FUNCTION_BLOCK Stage13 (* Template for a Basic Function Block Type *)
  (* Standard: 61499-2 *)
  (* Version 1.0, 2021-06-20, HP *)
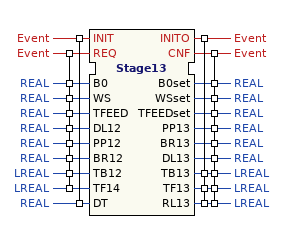
  EVENT_INPUT
    INIT WITH DT; (* Initialization Request *)
    REQ WITH B0, WS, TFEED, DL12, PP12, BR12, TB12, TF14; (* Normal Execution Request *)
  END_EVENT
  EVENT_OUTPUT
    INITO WITH TB13, TF13, RL13; (* Initialization Confirm *)
    CNF WITH TB13, DL13, TF13, BR13, PP13, TFEEDset, B0set, WSset, RL13; (* Execution Confirmation *)
  END_EVENT
  VAR_INPUT
    B0 : REAL;
    WS : REAL;
    TFEED : REAL;
    DL12 : REAL;
    PP12 : REAL;
    BR12 : REAL;
    TB12 : LREAL;
    TF14 : LREAL;
    DT : REAL;
  END_VAR
  VAR_OUTPUT
    B0set : REAL;
    WSset : REAL;
    TFEEDset : REAL;
    PP13 : REAL;
    BR13 : REAL;
    DL13 : REAL;
    TB13 : LREAL;
    TF13 : LREAL;
    RL13 : LREAL;
  END_VAR
  VAR
    AB : REAL; (* internal variabel *)
    UU : REAL;
    TREF : REAL;
    AD : REAL;
    AHC : REAL;
    AHR : REAL;
    AS : REAL;
    REC : REAL;
    WN : REAL;
    WN_1 : REAL;
    XKN : REAL;
    C1 : REAL;
    HS : REAL;
    G : REAL;
    W1 : REAL;
    TFREC : REAL;
    TS : REAL;
    DTS : REAL;
    TF13_last : REAL;
    RL13_last : REAL;
    TB13_last : REAL;
    USS : REAL;
    RHOB : REAL;
    CPB : REAL;
    CPF : REAL;
    FMW : REAL;
    HLV : REAL;
    HV : REAL;
    BPR : REAL;
    FMC : REAL;
    U : REAL;
    A : REAL;
    B : REAL;
    C : REAL;
    D1 : REAL;
    d : REAL;
    a : REAL;
    A1 : REAL;
    A2 : REAL;
    A3 : REAL;
    A4 : REAL;
    A5 : REAL;
    A6 : REAL;
    p : REAL;
    q : REAL;
    TC : REAL;
    PC : REAL;
    DTB13 : REAL;
    DEN13 : REAL;
    DH13 : REAL;
    DP13 : REAL;
    DPDH13 : REAL;
    DT13 : REAL;
    m : REAL;
    n : REAL;
    VR13 : REAL;
    DELTA13 : REAL;
    DELTA35 : REAL;
    DELTA57 : REAL;
    DELTA13_last : REAL;
    DELTA35_last : REAL;
    DELTA57_last : REAL;
  END_VAR
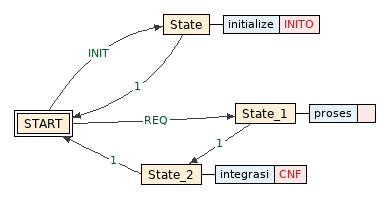
  EC_STATES
    START; (* Initial State *)
    State : initialize -> INITO;
    State_1 : proses;
    State_2 : integrasi -> CNF;
  END_STATES
  EC_TRANSITIONS
    START TO State := INIT;
    State TO START := 1;
    START TO State_1 := REQ;
    State_1 TO State_2 := 1;
    State_2 TO START := 1;
  END_TRANSITIONS
  ALGORITHM initialize IN ST: (* Initialization algorithm *)
TREF :=273.15;
AB :=57.2727;
AHC :=4069.2;
AHR :=2639.7;
AS :=3225.7;
REC :=0.0;
//TF2:=TF2;

//TFEED :=TFEED1+TREF;
 //TS:=TS1+TREF;
WN :=3.0;
XKN :=0.68;
HS:=0.11;
G :=9.81;
W1 :=0.50;

RL13 := 0.592736417366111;
TB13 := 332.856791580679;
TF13 := 329.218147337666;
TF14 := 326.857347111076;



RL13_last :=RL13;
TB13_last :=TB13;
TF13_last :=TF13;
  END_ALGORITHM
  ALGORITHM proses IN ST: (* kalkulasi *)
UU := TFEED;
U :=UU;

USS :=49.767;
C1 :=0.625;
RHOB :=1032.4; //maassa jenis brine
CPB :=1.00; //heatcapacity Brine
CPF :=1.00; //heat capacity feed
FMW :=23654.0;
HLV :=563.7959;
HV :=625.1971;
BPR :=2.192;
FMC :=34736.09;
//U :=UU; //feed temp



///  Calculate the physical properties

//A :=3.2437814;
//B :=5.86826*0.001;
//C :=1.1702379*0.00000001;
//D1 :=2.1878462*0.001;
//TC :=647.27;
//PC :=218.167;


A1 :=3.2437814;
A2:=5.86826*0.001;
A3:=1.1702379*0.00000001;
A4 :=2.1878462*0.001;
A5 :=647.27;
A6 :=218.167;

DTB13 :=A5-TB13;
DEN13 :=(A1+A2*DTB13+A3*DTB13*DTB13*DTB13)/(1+A4*DTB13)*DTB13/TB13;
p:=DEN13;
q:=10.0;
PP13 :=A6/(EXPT(q, p));

// calculate the brine flow rates
DP13:=PP12-PP13;
DH13:=RL13-C1*HS;
DPDH13 :=DP13*101000+G*RHOB*DH13;
m:=DPDH13*RHOB;
n:=0.5;
BR13 :=WN*XKN*RL13*(EXPT(m, n));
BR13 :=BR13*60.0/1000.0;

// calculate the vapor flow rates

DT13 :=TB13-BPR/1.8-(TF14+TF13)*0.5;
VR13:=U*AHC*DT13/HLV/1000.0;
DL13 :=DL12+VR13;


//// state equation
DELTA13 :=(BR12-BR13-VR13)*1000.0/RHOB/AB;
DELTA35 :=((BR12*CPB*(TB12-TB13))-VR13*(HV-CPB*(TB13-TREF)))*1000.0/AB/RHOB/CPB/RL13;
DELTA57 :=(B0*CPF*(TF14-TF13)*1000+(U*AHC*DT13))/FMW/CPF;
  END_ALGORITHM
  ALGORITHM integrasi IN ST: (* new algorithm *)
B0set:=B0;
WSset:=WS ;
TFEEDset:=TFEED;
//integrasi
RL13 := (DELTA13 + DELTA13_last)*0.5*DT + RL13_last;
DELTA13_last :=DELTA13 ;
RL13_last :=RL13;

TB13:= (DELTA35 + DELTA35_last)*0.5*DT + TB13_last;
DELTA35_last :=DELTA35 ;
TB13_last:=TB13;

TF13 := (DELTA57 + DELTA57_last)*0.5*DT + TF13_last;
DELTA57_last :=DELTA57 ;
TF13_last :=TF13;
  END_ALGORITHM
END_FUNCTION_BLOCK
